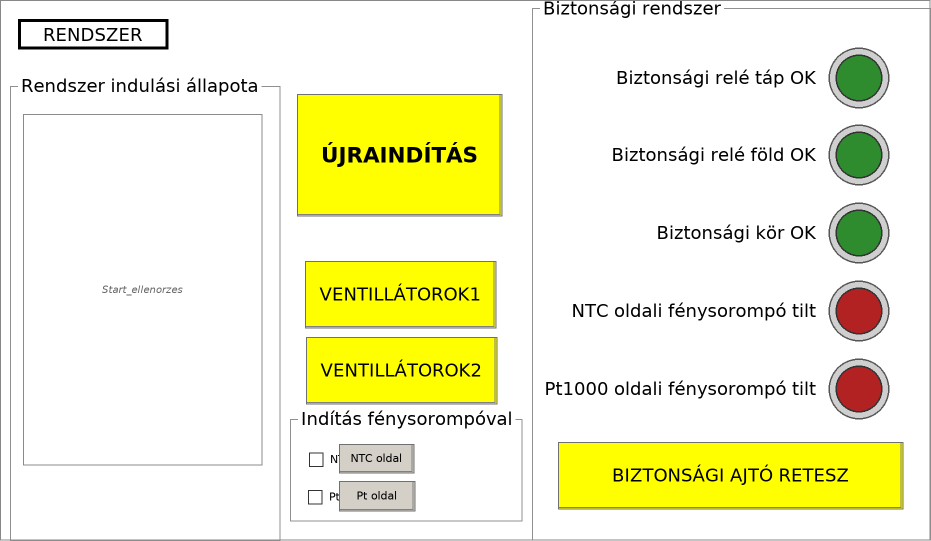
VISUALIZATION Rendszerinditas  // 931x541
    RoundedRectangle (18,19 150x30)
    Label (18,20 150x30), "RENDSZER"
    Button (297,94 205x122), "ÚJRAINDÍTÁS"
        OnMouseUp: execute { INIT.bRestart:=TRUE; }
    GroupBox (10,78 270x463), "Rendszer indulási állapota"
        Frame (13,36 239x351)
            shows Start_ellenorzes()
    GroupBox (532,0 399x540), "Biztonsági rendszer"
        Button (26,442 345x67), "BIZTONSÁGI AJTÓ RETESZ", pressed state: GVL.bBiztonsagiZarBe
            OnMouseClick: execute {
                IF GVL.bBiztonsagiZarBe=TRUE THEN
                	WHILE NOT (ROBOTREMOTE.sRobotCommand='') DO
                		;
                	END_WHILE
                	ROBOTREMOTE.sRobotCommand := 'Pause';
                	ROBOTREMOTE.bRobotCommandSend := TRUE;
                ELSE
                	WHILE NOT (ROBOTREMOTE.sRobotCommand='') DO
                		;
                	END_WHILE
                	ROBOTREMOTE.sRobotCommand := 'Continue';
                	ROBOTREMOTE.bRobotCommandSend := TRUE;
                END_IF
                GVL.bBiztonsagiZarBe:=NOT GVL.bBiztonsagiZarBe;
            }
        Lamp1 (292,43 70x70), variable: GVL.bBiztonsagiTap, style: Lamp-Lamp1-Green
        Label (17,63 270x30), "Biztonsági relé táp OK"
        Lamp1 (292,120 70x70), variable: NOT GVL.bBiztonsagiFold, style: Lamp-Lamp1-Green
        Label (17,140 270x30), "Biztonsági relé föld OK"
        Lamp1 (292,198 70x70), variable: (GVL.bBiztonsagiTap AND NOT GVL.bBiztonsagiFold) OR (NOT GVL.bBiztonsagiTap AND GVL.bBiztonsagiFold), style: Lamp-Lamp1-Green
        Label (17,218 270x30), "Biztonsági kör OK"
        Lamp1 (292,276 70x70), variable: NOT GVL.bFenysorompoNTC, style: Lamp-Lamp1-Red
        Label (17,296 270x30), "NTC oldali fénysorompó tilt"
        Lamp1 (292,354 70x70), variable: NOT GVL.bFenysorompoPt, style: Lamp-Lamp1-Red
        Label (17,374 270x30), "Pt1000 oldali fénysorompó tilt"
    Button (305,261 191x67), "VENTILLÁTOROK1", pressed state: GVL.bVentillatorok1Be
        toggle GVL.bVentillatorok1Be
    Button (306,337 191x67), "VENTILLÁTOROK2", pressed state: GVL.bVentillatorok2Be
        toggle GVL.bVentillatorok2Be
    GroupBox (290,411 232x110), "Indítás fénysorompóval"
        Checkbox (16,71 95x30), "Pt oldal", variable: GVL.bPtInditasFenysorompoval, input disabled if: TRUE
        Checkbox (17,34 94x29), "NTC oldal", variable: GVL.bNTCInditasFenysorompoval, input disabled if: TRUE
        Button (49,33 75x29), "NTC oldal", pressed state: GVL.bNTCInditasFenysorompoval
            toggle GVL.bNTCInditasFenysorompoval
            OnMouseUp: execute { AUTOMATA.iState:=102; }
        Button (49,70 76x30), "Pt oldal", pressed state: GVL.bPtInditasFenysorompoval
            toggle GVL.bPtInditasFenysorompoval
            OnMouseUp: execute { AUTOMATA.iState2:=103; }
END_VISUALIZATION

(* stored: Version 1.1.0.1, ProductVersion 3.1.4024.11
   Visu Rendszerinditas: Id {b0cd0b2d-9d58-463f-9c42-85f74b6e7dff} *)
